// TIA Portal V16 export
// export: Created 2024-09-05T17:39:13.8703633Z, ExportSetting WithDefaults, DisplayName Totally Integrated Automation Portal, DisplayVersion V16 Update 6, DisplayName TIA Portal Version Control Interface, DisplayVersion V16 Update 2, DisplayName TIA Portal Openness, DisplayVersion V16 Update 6, DisplayName STEP 7 Professional, DisplayVersion V16 Update 6, DisplayName STEP 7 Safety, DisplayVersion V16, DisplayName WinCC Advanced, DisplayVersion V16 Update 6
DATA_BLOCK "DB_Devices_Instance"   // DB5100
VERSION : 0.1
// stored: AutoNumber true, DBAccessibleFromOPCUA true, InstanceOfName FB_Devices, InstanceOfType FB
"FB_Devices"
   // VAR
   //    ServiceDoors_Instance_1 { S7_SetPoint := 'True'} : "serviceDoor";
   //    ServiceDoors_Instance_2 { S7_SetPoint := 'True'} : "serviceDoor";
   //    R_TRIG_Instance { S7_SetPoint := 'True'} : R_TRIG;
   //    HydraulicActive { S7_SetPoint := 'True'} : Bool := FALSE;
   //    HydraulicActiveOffMem : Bool := FALSE;
   //    HydraulicOnMem : Bool := FALSE;
   //    IEC_Timer_0_Instance { S7_SetPoint := 'True'} : TON_TIME;
   //    IEC_Timer_0_Instance_1 { S7_SetPoint := 'True'} : TON_TIME;
   //    FB_TurnTable_Instance { S7_SetPoint := 'True'} : "FB_TurnTable";
   //    F_TRIG_Instance { S7_SetPoint := 'True'} : F_TRIG;
   //    edges { S7_SetPoint := 'True'} : Array[1..6] of Bool;
   //    ManualCommandOld : Int := 0;
   //    R_TRIG_Instance_1 { S7_SetPoint := 'True'} : R_TRIG;
   //    R_TRIG_Instance_2 { S7_SetPoint := 'True'} : R_TRIG;
   //    R_TRIG_Instance_3 { S7_SetPoint := 'True'} : R_TRIG;
   //    R_TRIG_Instance_4 { S7_SetPoint := 'True'} : R_TRIG;
   //    R_TRIG_Instance_6 { S7_SetPoint := 'True'} : R_TRIG;
   //    R_TRIG_Instance_7 { S7_SetPoint := 'True'} : R_TRIG;
   //    R_TRIG_Instance_8 { S7_SetPoint := 'True'} : R_TRIG;
   //    R_TRIG_Instance_5 { S7_SetPoint := 'True'} : R_TRIG;
   //    edgesFitting : Array[1..4] of Bool;
   //    R_TRIG_V240Wp { S7_SetPoint := 'True'} : R_TRIG;
   //    R_TRIG_V240Bp { S7_SetPoint := 'True'} : R_TRIG;
   //    ReaderKeyence_Instance { S7_SetPoint := 'True'} : "ReaderKeyence";
   //    IEC_Timer_0_Instance_2 { S7_SetPoint := 'True'} : TON_TIME;
   //    FriedrichUnit1_Instance { S7_SetPoint := 'True'} : "FriedrichUnit";
   //    FriedrichUnit2_Instance { S7_SetPoint := 'True'} : "FriedrichUnit";
   //    Trig1 { S7_SetPoint := 'True'} : R_TRIG;
   //    Trig2 { S7_SetPoint := 'True'} : R_TRIG;
   //    Trig3 { S7_SetPoint := 'True'} : R_TRIG;
   //    Trig4 { S7_SetPoint := 'True'} : R_TRIG;
   //    Camera_CAM1 { S7_SetPoint := 'True'} : "Camera";
   //    Camera_CAM2 { S7_SetPoint := 'True'} : "Camera";
   //    Camera_CAM3 { S7_SetPoint := 'True'} : "Camera";
   //    Camera_CAM4 { S7_SetPoint := 'True'} : "Camera";
   //    RivetingCycleLeft_Instance { S7_SetPoint := 'True'} : "RivetingCycle";
   //    RivetingCycleRight_Instance { S7_SetPoint := 'True'} : "RivetingCycle";
   // END_VAR
BEGIN
   ServiceDoors_Instance_1.iButtonOpen := FALSE;
   ServiceDoors_Instance_1.iButtonLock := FALSE;
   ServiceDoors_Instance_1.iSequenceStoped := TRUE;
   ServiceDoors_Instance_1.iSafetyOK := TRUE;
   ServiceDoors_Instance_1.iDoorClosed := TRUE;
   ServiceDoors_Instance_1.qStopSequence := FALSE;
   ServiceDoors_Instance_1.qUnlock := FALSE;
   ServiceDoors_Instance_1.qLightOpen := FALSE;
   ServiceDoors_Instance_1.qLightLock := FALSE;
   ServiceDoors_Instance_1.stopRequest := FALSE;
   ServiceDoors_Instance_2.iButtonOpen := FALSE;
   ServiceDoors_Instance_2.iButtonLock := FALSE;
   ServiceDoors_Instance_2.iSequenceStoped := TRUE;
   ServiceDoors_Instance_2.iSafetyOK := TRUE;
   ServiceDoors_Instance_2.iDoorClosed := TRUE;
   ServiceDoors_Instance_2.qStopSequence := FALSE;
   ServiceDoors_Instance_2.qUnlock := FALSE;
   ServiceDoors_Instance_2.qLightOpen := FALSE;
   ServiceDoors_Instance_2.qLightLock := FALSE;
   ServiceDoors_Instance_2.stopRequest := FALSE;
   R_TRIG_Instance.CLK := FALSE;
   R_TRIG_Instance.Q := FALSE;
   R_TRIG_Instance.Stat_Bit := FALSE;
   IEC_Timer_0_Instance.PT := T#0MS;
   IEC_Timer_0_Instance.IN := FALSE;
   IEC_Timer_0_Instance_1.PT := T#0MS;
   IEC_Timer_0_Instance_1.IN := FALSE;
   FB_TurnTable_Instance.iTurnTableInputs := 16#0000;
   FB_TurnTable_Instance.iPower := FALSE;
   FB_TurnTable_Instance.iSafety := FALSE;
   FB_TurnTable_Instance.iReset := FALSE;
   FB_TurnTable_Instance.iErrorReset := FALSE;
   FB_TurnTable_Instance.iManualMode := TRUE;
   FB_TurnTable_Instance.iAutomaticMode := FALSE;
   FB_TurnTable_Instance.iTurnTableInSafetyPosition := TRUE;
   FB_TurnTable_Instance.qTurnTableOutputs := 16#0000;
   FB_TurnTable_Instance.qeCommunication := FALSE;
   FB_TurnTable_Instance.qeTurnTablePosition := FALSE;
   FB_TurnTable_Instance.qeTurnTableSafetyPosition := FALSE;
   FB_TurnTable_Instance.qeTimeout := FALSE;
   FB_TurnTable_Instance.qePositionRunOver := FALSE;
   FB_TurnTable_Instance.qeSafety := FALSE;
   FB_TurnTable_Instance.qeSumError := FALSE;
   FB_TurnTable_Instance.qeSumWarning := FALSE;
   FB_TurnTable_Instance.Edges.Enabled := FALSE;
   FB_TurnTable_Instance.Edges.IndexerInPosition := TRUE;
   FB_TurnTable_Instance.TONs.tDelayCommunication.PT := T#0MS;
   FB_TurnTable_Instance.TONs.tDelayCommunication.IN := FALSE;
   FB_TurnTable_Instance.TONs.tDelayPositionError.PT := T#3S;
   FB_TurnTable_Instance.TONs.tDelayPositionError.IN := FALSE;
   FB_TurnTable_Instance.TONs.tDelayErrorReset.PT := T#0MS;
   FB_TurnTable_Instance.TONs.tDelayErrorReset.IN := FALSE;
   FB_TurnTable_Instance.RetentiveData.LastDirection := FALSE;
   FB_TurnTable_Instance.Commands.ReadyToJogCW := FALSE;
   FB_TurnTable_Instance.Commands.JogCW := FALSE;
   FB_TurnTable_Instance.Commands.ReadyToJogCCW := FALSE;
   FB_TurnTable_Instance.Commands.JogCCW := FALSE;
   FB_TurnTable_Instance.Commands.ReadyToStartCW := FALSE;
   FB_TurnTable_Instance.Commands.StartCW := FALSE;
   FB_TurnTable_Instance.Commands.ReadyToStartCCW := FALSE;
   FB_TurnTable_Instance.Commands.StartCCW := FALSE;
   F_TRIG_Instance.CLK := FALSE;
   F_TRIG_Instance.Q := FALSE;
   F_TRIG_Instance.Stat_Bit := FALSE;
   edges[1..6] := FALSE;
   R_TRIG_Instance_1.CLK := FALSE;
   R_TRIG_Instance_1.Q := FALSE;
   R_TRIG_Instance_1.Stat_Bit := FALSE;
   R_TRIG_Instance_2.CLK := FALSE;
   R_TRIG_Instance_2.Q := FALSE;
   R_TRIG_Instance_2.Stat_Bit := FALSE;
   R_TRIG_Instance_3.CLK := FALSE;
   R_TRIG_Instance_3.Q := FALSE;
   R_TRIG_Instance_3.Stat_Bit := FALSE;
   R_TRIG_Instance_4.CLK := FALSE;
   R_TRIG_Instance_4.Q := FALSE;
   R_TRIG_Instance_4.Stat_Bit := FALSE;
   R_TRIG_Instance_6.CLK := FALSE;
   R_TRIG_Instance_6.Q := FALSE;
   R_TRIG_Instance_6.Stat_Bit := FALSE;
   R_TRIG_Instance_7.CLK := FALSE;
   R_TRIG_Instance_7.Q := FALSE;
   R_TRIG_Instance_7.Stat_Bit := FALSE;
   R_TRIG_Instance_8.CLK := FALSE;
   R_TRIG_Instance_8.Q := FALSE;
   R_TRIG_Instance_8.Stat_Bit := FALSE;
   R_TRIG_Instance_5.CLK := FALSE;
   R_TRIG_Instance_5.Q := FALSE;
   R_TRIG_Instance_5.Stat_Bit := FALSE;
   edgesFitting[1..4] := FALSE;
   R_TRIG_V240Wp.CLK := FALSE;
   R_TRIG_V240Wp.Q := FALSE;
   R_TRIG_V240Wp.Stat_Bit := FALSE;
   R_TRIG_V240Bp.CLK := FALSE;
   R_TRIG_V240Bp.Q := FALSE;
   R_TRIG_V240Bp.Stat_Bit := FALSE;
   ReaderKeyence_Instance."I_address_Read Data 128Byte" := 697;
   ReaderKeyence_Instance."Q_address_Operation instruction Control Bits" := 699;
   ReaderKeyence_Instance."Q_address_Parameter Bank Number" := 701;
   ReaderKeyence_Instance.iReset := FALSE;
   ReaderKeyence_Instance.ResultData[1..128] := ' ';
   ReaderKeyence_Instance.ResultDataReadyCountOld := 0;
   ReaderKeyence_Instance.R_TRIG_Instance.CLK := FALSE;
   ReaderKeyence_Instance.R_TRIG_Instance.Q := FALSE;
   ReaderKeyence_Instance.R_TRIG_Instance.Stat_Bit := FALSE;
   ReaderKeyence_Instance.IEC_Timer_0_Instance.PT := T#0MS;
   ReaderKeyence_Instance.IEC_Timer_0_Instance.IN := FALSE;
   IEC_Timer_0_Instance_2.PT := T#0MS;
   IEC_Timer_0_Instance_2.IN := FALSE;
END_DATA_BLOCK
